// TwinCAT 3 PLC project plc
// ProgramVersion: 3.1.4024.0
// libraries:
//   Tc2_Standard, * (Beckhoff Automation GmbH)
//   Tc2_System, * (Beckhoff Automation GmbH)
//   Tc3_JsonXml, * (Beckhoff Automation GmbH)
//   Tc3_Module, * (Beckhoff Automation GmbH)
// project tree:
//   / PlcTask.TcTTO (not stored)
//   POUs/ FB_ReadJsonReal.TcPOU, FB_SaveFile.TcPOU, MAIN.TcPOU
// real-time tasks:
//   TASK PlcTask: cycle T#10ms, priority 20, ADS port 350

// ---- POUs/FB_ReadJsonReal.TcPOU
FUNCTION_BLOCK FB_ReadJsonReal
VAR_INPUT
	Member:STRING;
	sPath:STRING;
END_VAR
VAR_OUTPUT
	fReadValue:LREAL;
	ReadDone:BOOL;
END_VAR
VAR
	nState: INT:=0;
	fbJsonDomParser:FB_JsonDomParser;
	ErrorCode :HRESULT;
	jSonProp :SJsonValue;
	jsonRoot :SJsonValue;
	bLoadDocument:BOOL;
END_VAR


CASE nState OF
	00: //Idle
		bLoadDocument:=FALSE;
		nState:=10;
		
	10: //Load the document
		bLoadDocument:=TRUE;
		fbJsonDomParser.LoadDocumentFromFile(sPath,bLoadDocument, hrErrorCode =>ErrorCode);
		IF ErrorCode = S_OK THEN
		nState:=20;
		END_IF
	
	20: //Read the desired values
		jsonRoot :=fbJsonDomParser.GetDocumentRoot();
		jSonProp := fbJsonDomParser.FindMember(jsonRoot,Member);
		IF (jsonProp<>0) THEN
			fReadValue := fbJsonDomParser.GetDouble(jSonProp);
			ReadDone:=TRUE;
		ELSE 
			fReadValue := -999999;
		END_IF
		
END_CASE

END_FUNCTION_BLOCK

// ---- POUs/FB_SaveFile.TcPOU
FUNCTION_BLOCK FB_SaveFile
VAR_INPUT
	sPath:STRING;
	AmsNetId:STRING;
	sBuffer:STRING(1024);
END_VAR
VAR_OUTPUT
	ErrorSaveFile:BOOL;
	SaveFileDone:BOOL;
END_VAR
VAR
	//Functions
	fbFileOpen   : FB_FileOpen;
    fbFileWrite  : FB_FileWrite;
    fbFileClose  : FB_FileClose;

	//Aux variables
	jsonDOC : SJsonValue;
	FileHandle :UINT;
	nState: INT:=0;
	
	bOpenExec:BOOL;
	bWriteExec:BOOL;
	bCloseExec:BOOL;
	
	nErrorIdOpen:UDINT;
	nErrorIdWrite:UDINT;
	nErrorIdClose:UDINT;
END_VAR

CASE nState OF
	00: //Idle
	bOpenExec:=FALSE;
	bWriteExec:=FALSE;
	bCloseExec:=FALSE;
	nState:=10;
		
	
	10://CreateFile
		bOpenExec:=TRUE;
		fbFileOpen(sNetId:=AmsNetId,sPathName := sPath,nMode := FOPEN_MODEWRITE OR FOPEN_MODETEXT,bExecute := bOpenExec);
		FileHandle :=fbFileOpen.hFile;
		IF NOT fbFileOpen.bError AND NOT fbFileOpen.bBusy THEN
		nState:=20;
		bOpenExec := FALSE;
		END_IF
		IF fbFileOpen.bError THEN
		nState :=999;			
		END_IF
		
	20: //Write the information
		bWriteExec:=TRUE;
		fbFileWrite(sNetId := AmsNetId,hFile := FileHandle,pWriteBuff := ADR(sBuffer),cbWriteLen := LEN(sBuffer),bExecute := bWriteExec);
		IF NOT fbFileWrite.bError AND NOT fbFileWrite.bBusy THEN
		bWriteExec :=FALSE;
		nState :=30;
		END_IF
		IF fbFileWrite.bError THEN
		nState :=999;			
		END_IF
		
	30: //Save the information and close the file
		bCloseExec:=TRUE;
		fbFileClose(sNetId:=AmsNetId, hFile := FileHandle, bExecute := bCloseExec);
		IF NOT fbFileClose.bError AND NOT fbFileClose.bBusy THEN
		FileHandle:=0;
		bCloseExec := FALSE;
		SaveFileDone:=TRUE;
		END_IF
		IF fbFileClose.bError THEN
		nState :=999;			
		END_IF
		
	999: //Error State
		ErrorSaveFile:=TRUE;
		nErrorIdOpen:=fbFileOpen.nErrId;
		nErrorIdWrite:=fbFileWrite.nErrId;
		nErrorIdClose:=fbFileClose.nErrId;	
	END_CASE

END_FUNCTION_BLOCK

// ---- POUs/MAIN.TcPOU
PROGRAM MAIN
VAR
	//Required functions
	fbJson:FB_JsonSaxWriter;
	fbSaveFile :FB_SaveFile;
	fbReadJsonReal :FB_ReadJsonReal;
	
	//Triggers for testing
	bTrigger: BOOL:=TRUE;
	bSave:BOOL;
	bLoadJsonFile:BOOL;
	
	//Buffer required to save the information in the json file. If a huge value is required, then change the string size here and in the FB_SaveFile
	sBuffer :STRING(255);
	
	//Random values for simulation
	r1:LREAL;
	r2:LREAL;
	r3:LREAL;

	//Variables to read the json file
	fSensor1Value :LREAL;
	fSensor2Value: LREAL;
	fSensor3Value: LREAL;
	fSensor4Value: LREAL;
	
END_VAR


//Trigger the following to gather random numbers
IF bTrigger THEN
	r1:=r1+(1.0/3.0);
	r2:=r2+(2.0/3.0);
	r3:=r3+(5.0/3.0);
	
	// JSON Object creation
	fbJson.StartObject(); //Open Bracket
		fbJson.AddKeyLreal('Sensor1',r1);
		fbJson.AddKeyLreal('Sensor2',r2);
		fbJson.AddKeyLreal('Sensor3',r3);
		fbJson.AddKeyLreal('Sensor4',r3);
	fbJson.EndObject(); //Close Bracket
	//Document creation
	sBuffer := fbJson.GetDocument();
	//Reset to get only one execution values
	fbJson.ResetDocument();
	
END_IF

//Save information, trigger bSave to create the file
IF bSave THEN
	fbSaveFile(sPath:='C:\TwinCAT\3.1\Boot\MyData.json',AmsNetId:='',sBuffer:=sBuffer);
	IF fbSaveFile.SaveFileDone AND NOT fbSaveFile.ErrorSaveFile THEN
	bSave:=FALSE;
	END_IF
END_IF

//Test, trigger bLoadJsonFile to read the information
IF bLoadJsonFile THEN
	fbReadJsonReal(Member:='Sensor1',sPath:='C:\TwinCAT\3.1\Boot\MyData.json',fReadValue=>);
	fSensor1Value:= fbReadJsonReal.fReadValue;
	
	fbReadJsonReal(Member:='Sensor2',sPath:='C:\TwinCAT\3.1\Boot\MyData.json',fReadValue=>);
	fSensor2Value:= fbReadJsonReal.fReadValue;
	
	fbReadJsonReal(Member:='Sensor3',sPath:='C:\TwinCAT\3.1\Boot\MyData.json',fReadValue=>);
	fSensor3Value:= fbReadJsonReal.fReadValue;
	
	fbReadJsonReal(Member:='Sensor4',sPath:='C:\TwinCAT\3.1\Boot\MyData.json',fReadValue=>);
	fSensor4Value:= fbReadJsonReal.fReadValue;
END_IF

END_PROGRAM
